(* IEC 61131-3 sources: RL_MAR/experiments/comparison/autoplc/results/deepseek-ai-DeepSeek-V3.2_20260508_111905/med_44, 1 file *)

(* ---- med_44_1.st ---- *)
FUNCTION_BLOCK DroneChargingStation
VAR_INPUT
    Drone1BatteryLevel : INT := 0; (* Battery level of Drone 1 (0-100%) *)
    Drone2BatteryLevel : INT := 0; (* Battery level of Drone 2 (0-100%) *)
    Drone3BatteryLevel : INT := 0; (* Battery level of Drone 3 (0-100%) *)
    ChargingTime : TIME := T#30s; (* Charging time required for each drone *)
END_VAR
VAR_OUTPUT
    Drone1Status : BOOL := FALSE; (* Status of Drone 1 *)
    Drone2Status : BOOL := FALSE; (* Status of Drone 2 *)
    Drone3Status : BOOL := FALSE; (* Status of Drone 3 *)
    ChargingStationStatus : BOOL := FALSE; (* Charging station status *)
    DroneDeployed : BOOL := FALSE; (* Indicates if a drone is deployed *)
END_VAR
VAR
    TimeRemaining : TIME := ChargingTime; (* Remaining charging time for the current charging operation *)
    bChargingStarted : BOOL := FALSE; (* Flag to track if charging has started *)
    bDeploymentTrigger : BOOL := FALSE; (* Internal deployment trigger *)
END_VAR

(* Main execution logic *)
IF NOT ChargingStationStatus THEN
    (* Charging station is not in use - check for drones needing charge *)
    IF NOT bChargingStarted THEN
        (* Check drone battery levels in order of priority *)
        IF (Drone1BatteryLevel < 20) AND NOT Drone1Status AND NOT Drone2Status AND NOT Drone3Status THEN
            Drone1Status := TRUE;
            ChargingStationStatus := TRUE;
            TimeRemaining := ChargingTime;
            bChargingStarted := TRUE;
        ELSIF (Drone2BatteryLevel < 20) AND NOT Drone1Status AND NOT Drone2Status AND NOT Drone3Status THEN
            Drone2Status := TRUE;
            ChargingStationStatus := TRUE;
            TimeRemaining := ChargingTime;
            bChargingStarted := TRUE;
        ELSIF (Drone3BatteryLevel < 20) AND NOT Drone1Status AND NOT Drone2Status AND NOT Drone3Status THEN
            Drone3Status := TRUE;
            ChargingStationStatus := TRUE;
            TimeRemaining := ChargingTime;
            bChargingStarted := TRUE;
        END_IF;
    END_IF;
ELSE
    (* Charging station is in use - manage charging timer *)
    IF TimeRemaining > T#0s THEN
        (* Decrement time remaining - assuming this is called in a cyclic task *)
        TimeRemaining := TimeRemaining - T#1ms; (* Adjust based on actual task cycle time *)
    ELSE
        (* Charging time has reached zero *)
        Drone1Status := FALSE;
        Drone2Status := FALSE;
        Drone3Status := FALSE;
        ChargingStationStatus := FALSE;
        bChargingStarted := FALSE;
        TimeRemaining := ChargingTime;
    END_IF;
END_IF;

(* Drone deployment management *)
(* Check if any deployed drone has critically low battery *)
IF DroneDeployed THEN
    IF (Drone1BatteryLevel < 10) OR (Drone2BatteryLevel < 10) OR (Drone3BatteryLevel < 10) THEN
        DroneDeployed := FALSE;
    END_IF;
END_IF;

(* Deployment trigger logic - requires external activation *)
(* This simulates an external deployment command *)
IF bDeploymentTrigger AND NOT DroneDeployed THEN
    DroneDeployed := TRUE;
    bDeploymentTrigger := FALSE;
END_IF;

END_FUNCTION_BLOCK
